// 隐含生成代码：这里只是对代码实现的建议
{noflow}
IF ptToTest=0 THEN
    ADSLOGSTR(ADSLOG_MSGTYPE_ERROR OR ADSLOG_MSGTYPE_STRING,'CheckPointer failed due to invalid address.','');
ELSIF iSize<=0 THEN
    ADSLOGSTR(ADSLOG_MSGTYPE_ERROR OR ADSLOG_MSGTYPE_STRING,'CheckPointer failed due to invalid size.','');
ELSIF iGran<=0 THEN
    ADSLOGSTR(ADSLOG_MSGTYPE_ERROR OR ADSLOG_MSGTYPE_STRING,'CheckPointer failed due to invalid granularity.','');
// -> Please note that the following memory area check is time consuming:
//ELSIF F_CheckMemoryArea(pData:=ptToTest,nSize:=DINT_TO_UDINT(iSize)) = E_TcMemoryArea.Unknown THEN
//    ADSLOGSTR(ADSLOG_MSGTYPE_ERROR OR ADSLOG_MSGTYPE_STRING,'CheckPointer failed due to unknown memory area.','');
END_IF
CheckPointer := ptToTest;
{flow}

END_FUNCTION

// ---- POUs/003_FB/43_implicit checks/CheckRangeSigned.TcPOU
// 隐含生成代码：不要编辑
FUNCTION CheckRangeSigned : DINT
VAR_INPUT
	value, lower, upper: DINT;
END_VAR

// 隐含生成代码：这里只是对代码实现的建议
{noflow}
IF (value < lower) THEN
	CheckRangeSigned := lower;
ELSIF(value > upper) THEN
	CheckRangeSigned := upper;
ELSE
	CheckRangeSigned := value;
END_IF
{flow}

END_FUNCTION

// ---- POUs/003_FB/43_implicit checks/CheckRangeUnsigned.TcPOU
// 隐含生成代码：不要编辑
FUNCTION CheckRangeUnsigned : UDINT
VAR_INPUT
	value, lower, upper: UDINT;
END_VAR

// 隐含生成代码：这里只是对代码实现的建议
{noflow}
IF (value < lower) THEN
	CheckRangeUnsigned := lower;
ELSIF(value > upper) THEN
	CheckRangeUnsigned := upper;
ELSE
	CheckRangeUnsigned := value;
END_IF
{flow}

END_FUNCTION

// ---- POUs/003_FB/53_RudongPump/08_PeristalticPumpFB/FB_RuDongPump_modbus_LABV.TcPOU
//{attribute 'tc_no_symbol'}
FUNCTION_BLOCK FB_RuDongPump_modbus_LABV
VAR_INPUT
	xExecute: BOOL;
	xAbort: BOOL;
	xResetRequest: BOOL;//匹配复位按钮 
	xRunILC				:BOOL;//蠕动泵运行条件
	dwTimeLimit: DWORD:=1;//[ms],1 => no invocation time limit
	dwTimeOut: DWORD;//[ms],0 => no executing time limit
	stPara       : RudongPump_Sys_Para;				
	xNeedConfigurePara		: BOOL := TRUE;//是否需要配置参数(默认是需要进行参数配置的)	
	stRunPara	:RudongPump_RunData;//运行参数	
	xAutoMode    : BOOL;//0:mannal 1:auto
	xIniting     : BOOL;//初始化过程中
	xDeviceRunning : BOOL;//工站单循环中
	rSpeedRatio  : REAL:=2.733;//根据泵头软管型号不同有变化
	sHmiError : STRING;
	xEStop : BOOL;
	stDeviceOpe	: RudongPump_Ope;//操作按钮
END_VAR
VAR_OUTPUT
	xDone: BOOL;(*完成条件满足*)
	xBusy: BOOL;(*动作正在执行*)
	xAborted: BOOL;(*指令被打断*)
	xRunning	:BOOL;//蠕动泵运行中
	eMobbusErrorID:UDINT;//modubs 报警信息
	xRudongPump_ERROR: BOOL;(*错误条件满足*)
	eERRORID: RudongPump_ERROR;(*错误码*)
	xRdyCmd : BOOL;
END_VAR
VAR_IN_OUT
		
END_VAR
VAR
{attribute 'tc_no_symbol'}
	eState: STATE;
{attribute 'tc_no_symbol'}
	_xDone: BOOL;
{attribute 'tc_no_symbol'}
	eCmd : RudongPump_CMD;//指令控制	
{attribute 'tc_no_symbol'}
	xFirstInvocation: BOOL := TRUE;	
{attribute 'tc_no_symbol'} 
	xTimeOut: BOOL;
{attribute 'tc_no_symbol'}
	xTimeLimit: BOOL;
{attribute 'tc_no_symbol'}
	tInvocationTimer , tOperationTimer : TON;
{attribute 'tc_no_symbol'}
	rFluVolumeSet   : REAL;//液量设定 0.0-99999.0 mL(0.1ml)
{attribute 'tc_no_symbol'}
	rRuntimeSet     : REAL;//运行时间设定 0.1-9999s(0.1s)
{attribute 'tc_no_symbol'}
	iCycleNumber		: INT;//重复次数
{attribute 'tc_no_symbol'}
	iModuleAdress		: INT;//灌装单元地址
{attribute 'tc_no_symbol'}
	iModuleSpeed		: REAL;//灌装单元速度
{attribute 'tc_no_symbol'}
	iModuleRealVolume	: REAL;//灌装实际液量	
{attribute 'tc_no_symbol'}
	_cmdStop  : BOOL;  
{attribute 'tc_no_symbol'}
	_tonTimeout , _tonCmdTimeout : TON;	
{attribute 'tc_no_symbol'}
  /// command execution
  _CmdExe : BOOL;
{attribute 'tc_no_symbol'}
  /// detect rising edge of command execution
  _rTrigCmdExe : R_TRIG;
{attribute 'tc_no_symbol'}	
  _rTrigCmdOrg   : R_TRIG;	
{attribute 'tc_no_symbol'}
	_diCmdState 	: DINT; 
{attribute 'tc_no_symbol'} 
  /// detect FltQuit rising edge
  _rTrigFltReset      : R_TRIG; 
{attribute 'tc_no_symbol'} 
  _tonDelay : TON; 
{attribute 'tc_no_symbol'}	
	_iConnectState : INT := 0;
{attribute 'tc_no_symbol'}	
	_connectTon : TON;
{attribute 'tc_no_symbol'}		
	_xConnectError : BOOL;
{attribute 'tc_no_symbol'}		
	_fResetCheck : F_TRIG;
{attribute 'tc_no_symbol'}		
	_rManual : R_TRIG;
{attribute 'tc_no_symbol'}		
	_fManual : F_TRIG;
{attribute 'tc_no_symbol'}		
	_xModeChange : BOOL;
{attribute 'tc_no_symbol'}		
	i : INT;
{attribute 'tc_no_symbol'}		
	_tonPulse : TON;//状态读取计时定时器
{attribute 'tc_no_symbol'}		
  _xCheckModbusRun : BOOL;//检测modbus是否处理总
{attribute 'tc_no_symbol'}	  
	_xConfigureParaOK : BOOL;//需要匹配参数是OK的
{attribute 'tc_no_symbol'}		
	_rStopCmdTrig : R_TRIG;
{attribute 'tc_no_symbol'}		
	_iActRunNumber : INT ;//当前运行的次数
{attribute 'tc_no_symbol'}		
	_wFluVolumeSetTemp : WORD;
{attribute 'tc_no_symbol'}		
	_wRuntimeSetTemp : WORD;
{attribute 'tc_no_symbol'}		
	_wSpeedSetTemp : WORD;	
{attribute 'tc_no_symbol'}	
 _tonDelay1:TON;
{attribute 'tc_no_symbol'}		
	_rSetSpeed : REAL;
{attribute 'tc_no_symbol'}		
	_wModuleSpeedSetTemp:WORD;
{attribute 'tc_no_symbol'}		
	_wModuleRealVolumeTemp:WORD;
{attribute 'tc_no_symbol'}		
	_rHMIControl : R_TRIG;
{attribute 'tc_no_symbol'}
	_iComNGCount:INT;
{attribute 'tc_no_symbol'}		
	dwTest1 : DWORD ;
{attribute 'tc_no_symbol'}		
	_iNGCount : INT;//NG 计数
{attribute 'tc_no_symbol'}		
	_rOperaTrig	:ARRAY [1..15] OF R_TRIG;
{attribute 'tc_no_symbol'}		
	k : INT;
{attribute 'tc_no_symbol'}		
	_bChannelNum , _bDiagData : BYTE;
{attribute 'tc_no_symbol'}		
	xAutomodeFlag	:BOOL;
{attribute 'tc_no_symbol'}		
	diStepOld:DINT;
{attribute 'tc_no_symbol'}			
	st_IOData : RudongPump_IOData;
{attribute 'tc_no_symbol'}		
	iPumpType	:INT;
{attribute 'tc_no_symbol'}	
	_xHMIOpe :BOOL;//是否有手动操作，是否有自动操作	
{attribute 'tc_no_symbol'}	
	 _xAutoOpe : BOOL;//是否有手动操作，是否有自动操作	
{attribute 'tc_no_symbol'}	
	_rInit	:R_TRIG;
{attribute 'tc_no_symbol'}		
	_first:BOOL;
{attribute 'tc_no_symbol'}				
	_aWrite_VAR: FB_MBWriteRegs; 
{attribute 'tc_no_symbol'}
//1:泵头型号；2:软管型号；3:启停控制	4:方向控制  5:全速运行  6:设定液量  7:时间设定  8:运行模式  9:重复次数		
//10:灌装单元地址  11:灌装单元速度  12:灌装单元启停  13:实际灌装量  14:灌装液量微调  15:恢复校准系数 			
  _aExecute : ARRAY[1..15] OF BOOL;    
{attribute 'tc_no_symbol'}	
  _aQuantity : ARRAY[1..15] OF WORD:=[1,1,1,1,1,2,2,1,1,1,2,1,2,1,1];  //寄存器个数   
{attribute 'tc_no_symbol'}	
  _aMBAddr : ARRAY[1..15] OF WORD:=[1000,1001,1008,1009,1010,1015,1018,1020,1023,2000,2001,2003,2004,2006,2007];  //起始地址   
{attribute 'tc_no_symbol'}		
  _aAddr : ARRAY[1..15,1..2] OF  INT;  //存放区域  
{attribute 'tc_no_symbol'}		
	_iChannelIndex:INT;
{attribute 'tc_no_symbol'}	
	_rxState:INT;
{attribute 'tc_no_symbol'}			
	_xBusy:BOOL;
END_VAR
VAR_TEMP
{attribute 'tc_no_symbol'}	
	xAgain: BOOL;
END_VAR

xAgain:=0;
ConnectAction();//触发通信连接功能连接
ACTMap();//IO Map
IF NOT _first THEN
	_first:=TRUE;
ELSE

//只有在运行的时候，才会检测是否有模式切换发生
IF eState <> STATE.DORMANT
THEN	
	IF _rManual.Q OR _fManual.Q
	THEN
		_xModeChange := TRUE;//通知系统有模式切换发生
	END_IF
ELSE
	_xModeChange := FALSE;//待机状态不触发模式切换
END_IF

//检测是否是初始化中，如果是的去切换模式
_rInit(CLK:= xIniting);
IF _rInit.Q
THEN
	eState := STATE.RESETING;
END_IF	

REPEAT
	CASE eState OF
		STATE.DORMANT:
				HandleDormantState(xAgain=> xAgain);
		STATE.EXECUTING:
				HandleExecutingState(xAgain=> xAgain);
		STATE.DONE:
				HandleDoneState(xAgain=> xAgain);
		STATE.INERROR:
				HandleErrorState(xAgain=> xAgain);
		STATE.ABORTING:
				HandleAbortingState(xAgain=> xAgain);
		STATE.ABORTED:
				HandleAbortedState(xAgain=> xAgain);
		STATE.RESETING:
				HandleResettingState(xAgain=> xAgain);
	END_CASE
UNTIL (xAgain=0)
END_REPEAT
END_IF


//判断是否处于当前流程的Done状态
xDone := _xDone AND xExecute;
//输出报错信息
CASE eERRORID OF 	
  RudongPump_ERROR.No_ERROR:
		sHmiError:='No_ERROR';	
  RudongPump_ERROR.FLT_PARA:
		sHmiError:='FLT_PARA';
  RudongPump_ERROR.FLT_CONNECT:
		sHmiError:='FLT_CONNECT';
  RudongPump_ERROR.FLT_RDYCMD:
		sHmiError:='FLT_RDYCMD';
	RudongPump_ERROR.FLT_CONFIGURE_PARA:
		sHmiError:='FLT_CONFIGURE_PARA';
	RudongPump_ERROR.FLT_FLUVOLUM_TIME_PARA:
		sHmiError:='FLT_FLUVOLUM_TIME_PARA';  
  RudongPump_ERROR.FLT_PUSH_TIMEOUT:
		sHmiError:='FLT_PUSH_TIMEOUT';
  RudongPump_ERROR.FLT_PULL_TIMEOUT:
		sHmiError:='FLT_PULL_TIMEOUT';
  RudongPump_ERROR.FLT_STOP_TIMEOUT:
		sHmiError:='FLT_STOP_TIMEOUT'; 
	RudongPump_ERROR.FLT_FULLSPEEDSTOP_TIMEOUT:
		sHmiError:='FLT_FULLSPEEDSTOP_TIMEOUT';
	RudongPump_ERROR.FLT_FULLSPEEDSTART_TIMEOUT:
		sHmiError:='FLT_FULLSPEEDSTART_TIMEOUT'; 
	RudongPump_ERROR.FLT_CMD_TIMEOUT:
		sHmiError:='FLT_CMD_TIMEOUT';
	RudongPump_ERROR.FLT_RUN_FALL:
		sHmiError:='FLT_RUN_FALL';
END_CASE
//手动自动操作检测
_xHMIOpe :=
			stDeviceOpe.xConfigure_Hmi OR 
			stDeviceOpe.xFullSpeedPull_Hmi OR 
			stDeviceOpe.xFullSpeedPush_Hmi OR 
			stDeviceOpe.xPull_Hmi[1] OR 
			stDeviceOpe.xPull_Hmi[2] OR 
			stDeviceOpe.xPull_Hmi[3] OR 
			stDeviceOpe.xPull_Hmi[4] OR 
			stDeviceOpe.xPull_Hmi[5] OR 			
			stDeviceOpe.xPumpCal_Hmi OR 
			stDeviceOpe.xPush_Hmi[1] OR 
			stDeviceOpe.xPush_Hmi[2] OR 
			stDeviceOpe.xPush_Hmi[3] OR 			
			stDeviceOpe.xPush_Hmi[4] OR 			
			stDeviceOpe.xPush_Hmi[5] OR 						
			stDeviceOpe.xResetCalcoeffCal_Hmi OR 
			stDeviceOpe.xStop_Hmi;
_xAutoOpe:=	
			stDeviceOpe.xConfigure_Auto OR 
            stDeviceOpe.xFullSpeedPull_Auto OR 
            stDeviceOpe.xFullSpeedPush_Auto OR 
            stDeviceOpe.xPull_Auto[1] OR 
            stDeviceOpe.xPull_Auto[2] OR 			
            stDeviceOpe.xPull_Auto[3] OR 			
            stDeviceOpe.xPull_Auto[4] OR 			
            stDeviceOpe.xPull_Auto[5] OR 			
            stDeviceOpe.xPumpCal_Auto OR 
            stDeviceOpe.xPush_Auto[1] OR 
            stDeviceOpe.xPush_Auto[2] OR 			
            stDeviceOpe.xPush_Auto[3] OR 			
            stDeviceOpe.xPush_Auto[4] OR 			
            stDeviceOpe.xPush_Auto[5] OR 						
            stDeviceOpe.xStop_Auto;

METHOD PROTECTED AbortAction
VAR_INPUT
END_VAR
VAR_OUTPUT
	xComplete: BOOL;
  eERRORID: RudongPump_ERROR;
END_VAR
(*
* Cleaning
* => abort all running operation
* => if an NBS.RudongPump_ERROR codition is reached, set eERRORID to a Value rather then NBS.RudongPump_ERROR.No_ERROR 
*)
xComplete:=1;
eERRORID:=RudongPump_ERROR.No_ERROR;
END_METHOD

ACTION ACTMap:

//1,泵头类型
	_aAddr[1,1]:= st_IOData.O_PumpType;
//2,软管类型	
	_aAddr[2,1] := st_IOData.O_HosePipeType;
//3,启停控制	
	_aAddr[3,1] := st_IOData.O_ControlSet;
//4,方向控制	
	_aAddr[4,1] := st_IOData.O_DirectionSet;
//5,全速控制	
	_aAddr[5,1] := st_IOData.O_FullSpeedControl;	
//6,液量设定	
	SysMemCpy(ADR(_aAddr[6,1]),ADR(st_IOData.O_FluVolumeSet),4);	
	_wFluVolumeSetTemp := TO_WORD(_aAddr[6,1]);
	_aAddr[6,1] := _aAddr[6,2];
	_aAddr[6,2] := TO_INT(_wFluVolumeSetTemp);
//7,运行时间设定	
	SysMemCpy(ADR(_aAddr[7,1]),ADR(st_IOData.O_RuntimeSet),4);
	_wRuntimeSetTemp := TO_WORD(_aAddr[7,1]);
	_aAddr[7,1] := _aAddr[7,2];
	_aAddr[7,2] := TO_INT(_wRuntimeSetTemp);	
//8,运行模式	
	_aAddr[8,1] := st_IOData.O_RunModeSet;
//9,重复次数	
	_aAddr[9,1] := st_IOData.O_CycleNumber;
//10,灌装单元地址
	_aAddr[10,1] := st_IOData.O_ModuleAddress;	
//11,灌装单元速度
	SysMemCpy(ADR(_aAddr[11,1]),ADR(st_IOData.O_ModuleSpeed),4);
	_wModuleSpeedSetTemp := TO_WORD(_aAddr[11,1]);
	_aAddr[11,1] := _aAddr[11,2];
	_aAddr[11,2] := TO_INT(_wModuleSpeedSetTemp);
//12,灌装单元启停
	_aAddr[12,1] := st_IOData.O_ModuleStart;	
//13,实际灌装液量
	SysMemCpy(ADR(_aAddr[13,1]),ADR(st_IOData.O_ModuleRealVolume),4);
	_wModuleRealVolumeTemp := TO_WORD(_aAddr[13,1]);
	_aAddr[13,1] := _aAddr[13,2];
	_aAddr[13,2] := TO_INT(_wModuleRealVolumeTemp);
//14,灌装液量微调
	_aAddr[14,1] := st_IOData.O_ModuleMicroReg;	
//15,恢复校准系数
	_aAddr[15,1] := st_IOData.O_ResetCalcoeff;		

xRunning:=stPara.xPumpRunSignal;//运行信号
iPumpType:=RudongPump_PumpType.LabV;//蠕动泵类型

_fResetCheck(CLK:=xResetRequest);
xRdyCmd := eState = STATE.DORMANT AND eERRORID = RudongPump_ERROR.No_ERROR;//检测是否允许指令控制(初始状态，没有报警发生)
(**********************************检测是否有模式切换********************************)
_rManual(CLK:=xAutoMode);
_fManual(CLK:=xAutoMode);
IF eState <> STATE.DORMANT//只有在运行的时候，才会检测是否有模式切换发生
THEN
	IF _rManual.Q OR _fManual.Q
	THEN
		_xModeChange := TRUE;//通知系统有模式切换发生
	END_IF	
END_IF
IF eState = STATE.DORMANT//要是待机模式下，切换模式，是不会起作用的
THEN
	_xModeChange := FALSE;
END_IF
(*************************检测配置参数是否匹配成功*********************************)
IF ( ( stRunPara.iPumpTypeSet = 0 OR stRunPara.iPumpTypeSet = 2 ) AND ( ( stRunPara.iHosePipeTypeSet >=13 AND stRunPara.iHosePipeTypeSet <=14 ) OR  
	 ( stRunPara.iHosePipeTypeSet >= 16 AND stRunPara.iHosePipeTypeSet <= 19 ) OR  stRunPara.iHosePipeTypeSet = 25 )) OR 
	 ( ( stRunPara.iPumpTypeSet = 1 OR stRunPara.iPumpTypeSet =3 ) AND ( stRunPara.iHosePipeTypeSet = 15 OR stRunPara.iHosePipeTypeSet = 24 ) ) OR 
	 ( ( stRunPara.iPumpTypeSet = 4 OR stRunPara.iPumpTypeSet = 5 ) AND (stRunPara.iHosePipeTypeSet >= 101 AND stRunPara.iHosePipeTypeSet <= 105 )) OR 
	 ( stRunPara.iPumpTypeSet = 6 AND (stRunPara.iHosePipeTypeSet = 15 OR stRunPara.iHosePipeTypeSet = 24 OR stRunPara.iHosePipeTypeSet = 35 OR stRunPara.iHosePipeTypeSet = 36)) OR 
	 ( stRunPara.iPumpTypeSet = 7 AND ( stRunPara.iHosePipeTypeSet = 14 OR stRunPara.iHosePipeTypeSet = 16 )) OR 
	 ( stRunPara.iPumpTypeSet = 8 AND stRunPara.iHosePipeTypeSet = 24 ) OR
   ( stRunPara.iPumpTypeSet = 17 AND (stRunPara.iHosePipeTypeSet = 15 OR stRunPara.iHosePipeTypeSet = 24 OR stRunPara.iHosePipeTypeSet = 35 OR stRunPara.iHosePipeTypeSet = 36) )	 
THEN
  _xConfigureParaOK := TRUE;
ELSE
	_xConfigureParaOK := FALSE;
END_IF
END_ACTION

METHOD PROTECTED CmdCalReset
VAR_OUTPUT
	xComplete: BOOL;
END_VAR
// return the real actual fault number
IF eERRORID <> RudongPump_ERROR.No_ERROR
THEN
  RETURN;  
END_IF

CASE _diCmdState OF	
		
		
	0://发送灌装系数复位指令
		_tonDelay(IN:= TRUE,pt:=T#20MS);//保证执行的是最新的一次
		st_IOData.O_ResetCalcoeff := 1	;	
		IF _tonDelay.Q
		THEN	
			_aExecute[15] := TRUE;//	
			//复位定时器
			_tonDelay(IN:=FALSE);
			_tonCmdTimeout(in:=FALSE);
			_tonTimeout(in:=FALSE);
			_diCmdState := _diCmdState+1;//切换状态
		END_IF
		
	1://等待灌装启动被响应
		_tonCmdTimeout(IN:= _aExecute[15],pt:=T#2S);
		IF NOT _aExecute[15]//
		THEN		
			_tonDelay(IN:=TRUE,PT:= T#50MS);
			IF _tonDelay.Q
			THEN
				_tonTimeout(in:=FALSE);
				_tonDelay(IN:=FALSE);
				_tonCmdTimeout(IN:= FALSE); 
				_diCmdState := _diCmdState+1;//切换状态
			END_IF	
		END_IF	
		IF _tonCmdTimeout.Q
		THEN
			eERRORID := RudongPump_ERROR.FLT_CMD_TIMEOUT;		
			_diCmdState := 999;
		END_IF	

	2://
		xComplete := TRUE; 
		
	ELSE
		;	
END_CASE
END_METHOD

METHOD PROTECTED CmdPumpCal
VAR_OUTPUT
	xComplete: BOOL;
END_VAR
// return the real actual fault number
IF eERRORID <> RudongPump_ERROR.No_ERROR
THEN
  RETURN;  
END_IF

CASE _diCmdState OF	
	0://检查参数	  	
		IF xNeedConfigurePara
		THEN
			_tonDelay(IN:= TRUE,pt:=T#25MS);//保证执行的是最新的一次
			st_IOData.O_RunModeSet := 2	;//打开定时定量模式
			IF _tonDelay.Q
			THEN	
				_aExecute[8] := TRUE;//启动夹紧控制数据发送	
				//复位定时器
				_tonDelay(IN:=FALSE);
				_tonCmdTimeout(in:=FALSE);
				_tonTimeout(in:=FALSE);
				_diCmdState := _diCmdState+1;//切换状态
			END_IF
		ELSE//直接启动就好
			//复位定时器
			_tonDelay(IN:=FALSE);
			_tonCmdTimeout(in:=FALSE);
			_tonTimeout(in:=FALSE);
			_diCmdState := 8;//切换状态
		END_IF	
		//检测流量转速是否在0.1rpm - 600rpm
		IF 	rRuntimeSet = 0 
		THEN 
			eERRORID := RudongPump_ERROR.FLT_FLUVOLUM_TIME_PARA;		
			_diCmdState := 999;
		ELSE
			_rSetSpeed := rFluVolumeSet * 60.0 / rSpeedRatio / rRuntimeSet;
			IF _rSetSpeed >= 0.1 AND _rSetSpeed <= 600
			THEN
				;
			ELSE
				eERRORID := RudongPump_ERROR.FLT_FLUVOLUM_TIME_PARA;		
				_diCmdState := 999;
			END_IF
		END_IF				
		
	1://等待定时定量模式被响应
		_tonCmdTimeout(IN:= _aExecute[8],pt:=T#2S);
		IF NOT _aExecute[8]//
		THEN		
			_tonDelay(IN:=TRUE,PT:= T#50MS);
			IF _tonDelay.Q
			THEN			
				_tonTimeout(in:=FALSE);
				_tonDelay(IN:=FALSE);
				_tonCmdTimeout(IN:= FALSE);    
				_diCmdState := _diCmdState+1;//切换状态
			END_IF	
		END_IF	
		IF _tonCmdTimeout.Q
		THEN
			eERRORID := RudongPump_ERROR.FLT_CMD_TIMEOUT;		
			_diCmdState := 999;
		END_IF


//发送虚假定量时间		
	2://定量时间设定		
		_tonDelay(IN:= TRUE,pt:=T#25MS);//保证执行的是最新的一次
		st_IOData.O_RuntimeSet := 200.0	;	//保证电机转速不会超
		IF _tonDelay.Q
		THEN	
			_aExecute[7] := TRUE;//启动夹紧控制数据发送	
			//复位定时器
			_tonDelay(IN:=FALSE);
			_tonCmdTimeout(in:=FALSE);
			_tonTimeout(in:=FALSE);
			_diCmdState := _diCmdState+1;//切换状态
		END_IF
	3://等待定量时间设定被响应
		_tonCmdTimeout(IN:= _aExecute[7],pt:=T#2S);
		IF NOT _aExecute[7]//
		THEN		
			_tonDelay(IN:=TRUE,PT:= T#50MS);
			IF _tonDelay.Q
			THEN			
				_tonTimeout(in:=FALSE);
				_tonDelay(IN:=FALSE);
				_tonCmdTimeout(IN:= FALSE);    
				_diCmdState := _diCmdState+1;//切换状态
			END_IF	
		END_IF	
		IF _tonCmdTimeout.Q
		THEN
			eERRORID := RudongPump_ERROR.FLT_CMD_TIMEOUT;		
			_diCmdState := 999;
		END_IF		
		
		
//传递液量参数		
	4://		
		_tonDelay(IN:= TRUE,pt:=T#25MS);//保证执行的是最新的一次
		st_IOData.O_FluVolumeSet := rFluVolumeSet	;	
		IF _tonDelay.Q
		THEN	
			_aExecute[6] := TRUE;//启动夹紧控制数据发送	
			//复位定时器
			_tonDelay(IN:=FALSE);
			_tonCmdTimeout(in:=FALSE);
			_tonTimeout(in:=FALSE);
			_diCmdState := _diCmdState+1;//切换状态
		END_IF	  
	5://等待流量设定结束
		_tonCmdTimeout(IN:= _aExecute[6],pt:=T#2S);
		IF NOT _aExecute[6]//
		THEN		
			_tonDelay(IN:=TRUE,PT:= T#50MS);
			IF _tonDelay.Q
			THEN			
				_tonTimeout(in:=FALSE);
				_tonDelay(IN:=FALSE);
				_tonCmdTimeout(IN:= FALSE);    
				_diCmdState := _diCmdState+1;//切换状态
			END_IF	
		END_IF	
		IF _tonCmdTimeout.Q
		THEN
			eERRORID := RudongPump_ERROR.FLT_CMD_TIMEOUT;		
			_diCmdState := 999;
		END_IF

//传递实际定量时间		
	6://定量时间设定		
		_tonDelay(IN:= TRUE,pt:=T#25MS);//保证执行的是最新的一次
		st_IOData.O_RuntimeSet := rRuntimeSet	;	
		IF _tonDelay.Q
		THEN	
			_aExecute[7] := TRUE;//启动夹紧控制数据发送	
			//复位定时器
			_tonDelay(IN:=FALSE);
			_tonCmdTimeout(in:=FALSE);
			_tonTimeout(in:=FALSE);
			_diCmdState := _diCmdState+1;//切换状态
		END_IF
		
	7://等待定量时间设定被响应
		_tonCmdTimeout(IN:= _aExecute[7],pt:=T#2S);
		IF NOT _aExecute[7]//
		THEN		
			_tonDelay(IN:=TRUE,PT:= T#50MS);
			IF _tonDelay.Q
			THEN			
				_tonTimeout(in:=FALSE);
				_tonDelay(IN:=FALSE);
				_tonCmdTimeout(IN:= FALSE);    
				_diCmdState := _diCmdState+1;//切换状态
			END_IF	
		END_IF	
		IF _tonCmdTimeout.Q
		THEN
			eERRORID := RudongPump_ERROR.FLT_CMD_TIMEOUT;		
			_diCmdState := 999;
		END_IF	
		
	8://方向设定		
		_tonDelay(IN:= ( eCmd = RudongPump_CMD.Cmd_CalPump ) ,pt:=T#20MS);//保证执行的是最新的一次
		st_IOData.O_DirectionSet := 1	;			
		IF _tonDelay.Q
		THEN	
			_aExecute[4] := TRUE;//启动夹紧控制数据发送	
			//复位定时器
			_tonDelay(IN:=FALSE);
			_tonCmdTimeout(in:=FALSE);
			_tonTimeout(in:=FALSE);
			_diCmdState := _diCmdState+1;//切换状态
		END_IF
		
	9://等待方向设定被响应
		_tonCmdTimeout(IN:= _aExecute[4],pt:=T#2S);
		IF NOT _aExecute[4]//
		THEN		
			_diCmdState := _diCmdState +1; 
			_tonDelay(IN:=FALSE);
			_tonCmdTimeout(in:=FALSE);
			_tonTimeout(in:=FALSE);
		END_IF	
		IF _tonCmdTimeout.Q
		THEN
			eERRORID := RudongPump_ERROR.FLT_CMD_TIMEOUT;		
			_diCmdState := 999;
		END_IF	
		
	10://重复次数设定		
		_tonDelay(IN:= TRUE,pt:=T#25MS);//保证执行的是最新的一次
		st_IOData.O_CycleNumber := iCycleNumber	;	
		IF _tonDelay.Q
		THEN	
			_aExecute[9] := TRUE;//启动夹紧控制数据发送	
			//复位定时器
			_tonDelay(IN:=FALSE);
			_tonCmdTimeout(in:=FALSE);
			_tonTimeout(in:=FALSE);
			_diCmdState := _diCmdState+1;//切换状态
		END_IF
		
	11://等待重复次数设定被响应
		_tonCmdTimeout(IN:= _aExecute[9],pt:=T#2S);
		IF NOT _aExecute[9]//
		THEN		
			_tonDelay(IN:=TRUE,PT:= T#50MS);
			IF _tonDelay.Q
			THEN
				_tonTimeout(in:=FALSE);
				_tonDelay(IN:=FALSE);
				_tonCmdTimeout(IN:= FALSE); 
				_diCmdState := _diCmdState+1;//切换状态
			END_IF	
		END_IF	
		IF _tonCmdTimeout.Q
		THEN
			eERRORID := RudongPump_ERROR.FLT_CMD_TIMEOUT;		
			_diCmdState := 999;
		END_IF		
		
	12://单元地址设定
		_tonDelay(IN:= TRUE,pt:=T#20MS);//保证执行的是最新的一次
		st_IOData.O_ModuleAddress := iModuleAdress	;
		//st_IOData.O_ModuleSpeed := iModuleSpeed	;	
		IF _tonDelay.Q
		THEN	
			_aExecute[10] := TRUE;//	
			//复位定时器
			_tonDelay(IN:=FALSE);
			_tonCmdTimeout(in:=FALSE);
			_tonTimeout(in:=FALSE);
			_diCmdState := _diCmdState+1;//切换状态
		END_IF
		
	13://等待单元地址设定被响应
	IF iPumpType=RudongPump_PumpType.DFPluse THEN	
		_tonCmdTimeout(IN:= _aExecute[10],pt:=T#2S);
		IF NOT _aExecute[10]//
		THEN		
			_tonDelay(IN:=TRUE,PT:= T#50MS);
			IF _tonDelay.Q
			THEN
				_tonTimeout(in:=FALSE);
				_tonDelay(IN:=FALSE);
				_tonCmdTimeout(IN:= FALSE); 
				_diCmdState := _diCmdState+1;//切换状态
			END_IF	
		END_IF	
		IF _tonCmdTimeout.Q
		THEN
			eERRORID := RudongPump_ERROR.FLT_CMD_TIMEOUT;		
			_diCmdState := 999;
		END_IF
	ELSE
		_diCmdState := 15;	
	END_IF	
		
	14://单元速度设定
	IF st_IOData.O_RunModeSet =1	THEN//如果是定量模式，需要设置速度
		_tonDelay(IN:= TRUE,pt:=T#20MS);//保证执行的是最新的一次
		st_IOData.O_ModuleSpeed := iModuleSpeed	;	
		IF _tonDelay.Q
		THEN	
			_aExecute[11] := TRUE;//	
			//复位定时器
			_tonDelay(IN:=FALSE);
			_tonCmdTimeout(in:=FALSE);
			_tonTimeout(in:=FALSE);
			_diCmdState := _diCmdState+1;//切换状态
		END_IF
	ELSE
		_diCmdState :=16;//如果是定时定量模式，则不需要设置速度
	END_IF	
	
	15://等待单元速度设定被响应
		_iNGCount :=0;
		_tonCmdTimeout(IN:= _aExecute[11],pt:=T#2S);
		IF NOT _aExecute[11]//
		THEN		
			_tonDelay(IN:=TRUE,PT:= T#50MS);
			IF _tonDelay.Q
			THEN
				_tonTimeout(in:=FALSE);
				_tonDelay(IN:=FALSE);
				_tonCmdTimeout(IN:= FALSE); 
				_diCmdState := _diCmdState+1;//切换状态
			END_IF	
		END_IF	
		IF _tonCmdTimeout.Q
		THEN
			eERRORID := RudongPump_ERROR.FLT_CMD_TIMEOUT;		
			_diCmdState := 999;
		END_IF		
		
	16://复位	
		st_IOData.O_ModuleStart := 0	;
		_aExecute[12] := FALSE;//		
		_diCmdState := _diCmdState+1;//切换状态
		
	17://灌装启动
		_tonDelay(IN:= TRUE,pt:=T#20MS);//保证执行的是最新的一次
		st_IOData.O_ModuleStart := 1	;	
		IF _tonDelay.Q
		THEN	
			_aExecute[12] := TRUE;//	
			//复位定时器
			_tonDelay(IN:=FALSE);
			_tonCmdTimeout(in:=FALSE);
			_tonTimeout(in:=FALSE);
			_diCmdState := _diCmdState+1;//切换状态
		END_IF
		
	18://等待灌装启动被响应
		_tonTimeout(in:=TRUE,pt:=T#30MS); 		
		_tonCmdTimeout(IN:= _aExecute[12],pt:=T#2S);
		IF stPara.xPumpRunSignal//一定要检测到泵运行
		THEN		
			_tonDelay(IN:=FALSE);
			_tonCmdTimeout(in:=FALSE);
			_diCmdState := _diCmdState +1; 
			_tonTimeout(in:=FALSE);	
		END_IF			
		IF _tonCmdTimeout.Q
		THEN
			eERRORID := RudongPump_ERROR.FLT_CMD_TIMEOUT;		
			_diCmdState := 999;
		END_IF
	IF _tonCmdTimeout.Q THEN
		_iNGCount := _iNGCount + 1;		
		IF _iNGCount <= 3
		THEN
			_tonDelay(IN:=FALSE);
			_tonCmdTimeout(IN:=FALSE);
			_tonTimeout(IN:=FALSE);
			_diCmdState := 15;//重新触发启动
		ELSE
			eERRORID := RudongPump_ERROR.FLT_PumpCal_TIMEOUT;					
			_diCmdState := 999;
		END_IF
	 END_IF		
		
	19://等待接液完成
		IF NOT stPara.xPumpRunSignal AND (stDeviceOpe.xPumpCal_Hmi OR stDeviceOpe.xPumpCal_Auto) AND NOT _xCheckModbusRun THEN
			_diCmdState := _diCmdState+1;//切换状态
		END_IF
		
	20://单元实际液量设定
		_tonDelay(IN:= TRUE,pt:=T#20MS);//保证执行的是最新的一次
		st_IOData.O_ModuleRealVolume := iModuleRealVolume	;	
		IF _tonDelay.Q
		THEN	
			_aExecute[13] := TRUE;//	
			//复位定时器
			_tonDelay(IN:=FALSE);
			_tonCmdTimeout(in:=FALSE);
			_tonTimeout(in:=FALSE);
			_diCmdState := _diCmdState+1;//切换状态
		END_IF
		
	21://等待单元实际液量设定被响应
		_tonCmdTimeout(IN:= _aExecute[13],pt:=T#2S);
		IF NOT _aExecute[13]//
		THEN		
			_tonDelay(IN:=TRUE,PT:= T#50MS);
			IF _tonDelay.Q
			THEN
				_tonTimeout(in:=FALSE);
				_tonDelay(IN:=FALSE);
				_tonCmdTimeout(IN:= FALSE); 
				_diCmdState := _diCmdState+1;//切换状态
			END_IF	
		END_IF	
		IF _tonCmdTimeout.Q
		THEN
			eERRORID := RudongPump_ERROR.FLT_CMD_TIMEOUT;		
			_diCmdState := 999;
		END_IF		

	22://
		xComplete := TRUE; 
		
	ELSE
		;	
END_CASE
END_METHOD

METHOD PROTECTED CmdRunAction
VAR_OUTPUT
	xComplete: BOOL;
END_VAR
// return the real actual fault number
IF eERRORID <> RudongPump_ERROR.No_ERROR
THEN
  RETURN;  
END_IF

CASE _diCmdState OF	
	0://传送力值和速度参数		  	
		IF xNeedConfigurePara
		THEN
			_tonDelay(IN:= TRUE,pt:=T#25MS);//保证执行的是最新的一次
			st_IOData.O_RunModeSet := 2	;//打开定时定量模式
			IF _tonDelay.Q
			THEN	
				_aExecute[8] := TRUE;//启动夹紧控制数据发送	
				//复位定时器
				_tonDelay(IN:=FALSE);
				_tonCmdTimeout(in:=FALSE);
				_tonTimeout(in:=FALSE);
				_diCmdState := _diCmdState+1;//切换状态
			END_IF
		ELSE//直接启动就好
			//复位定时器
			_tonDelay(IN:=FALSE);
			_tonCmdTimeout(in:=FALSE);
			_tonTimeout(in:=FALSE);
			_diCmdState := 12;//切换状态
		END_IF	
		//检测流量转速是否在0.1rpm - 600rpm
		IF 	rRuntimeSet = 0 
		THEN 
			eERRORID := RudongPump_ERROR.FLT_FLUVOLUM_TIME_PARA;		
			_diCmdState := 999;
		ELSE
			_rSetSpeed := rFluVolumeSet * 60.0 / rSpeedRatio / rRuntimeSet;
			IF _rSetSpeed >= 0.1 AND _rSetSpeed <= 600
			THEN
				;
			ELSE
				eERRORID := RudongPump_ERROR.FLT_FLUVOLUM_TIME_PARA;		
				_diCmdState := 999;
			END_IF
		END_IF				
		
	1://等待定时定量模式被响应
		_tonCmdTimeout(IN:= _aExecute[8],pt:=T#2S);
		IF NOT _aExecute[8]//
		THEN		
			_tonDelay(IN:=TRUE,PT:= T#50MS);
			IF _tonDelay.Q
			THEN			
				_tonTimeout(in:=FALSE);
				_tonDelay(IN:=FALSE);
				_tonCmdTimeout(IN:= FALSE);    
				_diCmdState := _diCmdState+1;//切换状态
			END_IF	
		END_IF	
		IF _tonCmdTimeout.Q
		THEN
			eERRORID := RudongPump_ERROR.FLT_CMD_TIMEOUT;		
			_diCmdState := 999;
		END_IF


//发送虚假定量时间		
	2://定量时间设定		
		_tonDelay(IN:= TRUE,pt:=T#25MS);//保证执行的是最新的一次
		st_IOData.O_RuntimeSet := 200.0	;	//保证电机转速不会超
		IF _tonDelay.Q
		THEN	
			_aExecute[7] := TRUE;//启动夹紧控制数据发送	
			//复位定时器
			_tonDelay(IN:=FALSE);
			_tonCmdTimeout(in:=FALSE);
			_tonTimeout(in:=FALSE);
			_diCmdState := _diCmdState+1;//切换状态
		END_IF
	3://等待定量时间设定被响应
		_tonCmdTimeout(IN:= _aExecute[7],pt:=T#2S);
		IF NOT _aExecute[7]//
		THEN		
			_tonDelay(IN:=TRUE,PT:= T#50MS);
			IF _tonDelay.Q
			THEN			
				_tonTimeout(in:=FALSE);
				_tonDelay(IN:=FALSE);
				_tonCmdTimeout(IN:= FALSE);    
				_diCmdState := _diCmdState+1;//切换状态
			END_IF	
		END_IF	
		IF _tonCmdTimeout.Q
		THEN
			eERRORID := RudongPump_ERROR.FLT_CMD_TIMEOUT;		
			_diCmdState := 999;
		END_IF		
		
		
//传递液量参数		
	4://传送力值和速度参数		
		_tonDelay(IN:= TRUE,pt:=T#25MS);//保证执行的是最新的一次
		st_IOData.O_FluVolumeSet := rFluVolumeSet	;	
		IF _tonDelay.Q
		THEN	
			_aExecute[6] := TRUE;//启动夹紧控制数据发送	
			//复位定时器
			_tonDelay(IN:=FALSE);
			_tonCmdTimeout(in:=FALSE);
			_tonTimeout(in:=FALSE);
			_diCmdState := _diCmdState+1;//切换状态
		END_IF	  
	5://等待流量设定结束
		_tonCmdTimeout(IN:= _aExecute[6],pt:=T#2S);
		IF NOT _aExecute[6]//
		THEN		
			_tonDelay(IN:=TRUE,PT:= T#50MS);
			IF _tonDelay.Q
			THEN			
				_tonTimeout(in:=FALSE);
				_tonDelay(IN:=FALSE);
				_tonCmdTimeout(IN:= FALSE);    
				_diCmdState := _diCmdState+1;//切换状态
			END_IF	
		END_IF	
		IF _tonCmdTimeout.Q
		THEN
			eERRORID := RudongPump_ERROR.FLT_CMD_TIMEOUT;		
			_diCmdState := 999;
		END_IF

//传递实际定量时间		
	6://定量时间设定		
		_tonDelay(IN:= TRUE,pt:=T#25MS);//保证执行的是最新的一次
		st_IOData.O_RuntimeSet := rRuntimeSet	;	
		IF _tonDelay.Q
		THEN	
			_aExecute[7] := TRUE;//启动夹紧控制数据发送	
			//复位定时器
			_tonDelay(IN:=FALSE);
			_tonCmdTimeout(in:=FALSE);
			_tonTimeout(in:=FALSE);
			_diCmdState := _diCmdState+1;//切换状态
		END_IF
		
	7://等待定量时间设定被响应
		_tonCmdTimeout(IN:= _aExecute[7],pt:=T#2S);
		IF NOT _aExecute[7]//
		THEN		
			_tonDelay(IN:=TRUE,PT:= T#50MS);
			IF _tonDelay.Q
			THEN			
				_tonTimeout(in:=FALSE);
				_tonDelay(IN:=FALSE);
				_tonCmdTimeout(IN:= FALSE);    
				_diCmdState := _diCmdState+1;//切换状态
			END_IF	
		END_IF	
		IF _tonCmdTimeout.Q
		THEN
			eERRORID := RudongPump_ERROR.FLT_CMD_TIMEOUT;		
			_diCmdState := 999;
		END_IF	
		
	8://方向设定		
		_tonDelay(IN:= ( eCmd = RudongPump_CMD.Cmd_Push OR eCmd = RudongPump_CMD.Cmd_Pull ) ,pt:=T#20MS);//保证执行的是最新的一次
		IF eCmd = RudongPump_CMD.Cmd_Push
		THEN
			st_IOData.O_DirectionSet := 1	;			
		END_IF
		IF eCmd = RudongPump_CMD.Cmd_Pull 
		THEN
			st_IOData.O_DirectionSet := 0	;			
		END_IF
		IF _tonDelay.Q
		THEN	
			_aExecute[4] := TRUE;//启动夹紧控制数据发送	
			//复位定时器
			_tonDelay(IN:=FALSE);
			_tonCmdTimeout(in:=FALSE);
			_tonTimeout(in:=FALSE);
			_diCmdState := _diCmdState+1;//切换状态
		END_IF
		
	9://等待方向设定被响应
		_tonCmdTimeout(IN:= _aExecute[4],pt:=T#2S);
		IF NOT _aExecute[4]//
		THEN		
			_diCmdState := _diCmdState +1; 
			_tonDelay(IN:=FALSE);
			_tonCmdTimeout(in:=FALSE);
			_tonTimeout(in:=FALSE);
		END_IF	
		IF _tonCmdTimeout.Q
		THEN
			eERRORID := RudongPump_ERROR.FLT_CMD_TIMEOUT;		
			_diCmdState := 999;
		END_IF	
		
	10://重复次数设定		
		_tonDelay(IN:= TRUE,pt:=T#25MS);//保证执行的是最新的一次
		st_IOData.O_CycleNumber := iCycleNumber	;	
		IF _tonDelay.Q
		THEN	
			_aExecute[9] := TRUE;//启动夹紧控制数据发送	
			//复位定时器
			_tonDelay(IN:=FALSE);
			_tonCmdTimeout(in:=FALSE);
			_tonTimeout(in:=FALSE);
			_diCmdState := _diCmdState+1;//切换状态
		END_IF
		
	11://等待重复次数设定被响应
		_tonCmdTimeout(IN:= _aExecute[9],pt:=T#2S);
		IF NOT _aExecute[9]//
		THEN		
			_tonDelay(IN:=TRUE,PT:= T#50MS);
			IF _tonDelay.Q
			THEN
				_tonTimeout(in:=FALSE);
				_tonDelay(IN:=FALSE);
				_tonCmdTimeout(IN:= FALSE); 
				_diCmdState := _diCmdState+1;//切换状态
			END_IF	
		END_IF	
		IF _tonCmdTimeout.Q
		THEN
			eERRORID := RudongPump_ERROR.FLT_CMD_TIMEOUT;		
			_diCmdState := 999;
		END_IF		
		
	12://启动设定		
		_tonDelay(IN:= TRUE ,pt:=T#25MS);//保证执行的是最新的一次	
		st_IOData.O_ControlSet := 1	;					
		IF _tonDelay.Q
		THEN	
			_aExecute[3] := TRUE;//启动夹紧控制数据发送	
			//复位定时器
			_tonDelay(IN:=FALSE);
			_tonCmdTimeout(in:=FALSE);
			_tonTimeout(in:=FALSE);
			_diCmdState := _diCmdState+1;//切换状态
		END_IF
		
	13://等待启动被响应
		_tonTimeout(in:=TRUE,pt:=T#4S); 		
		_tonCmdTimeout(IN:= _aExecute[3],pt:=T#2S);
		IF stPara.xPumpRunSignal//一定要检测到泵运行
		THEN		
			_tonDelay(IN:=FALSE);
			_tonCmdTimeout(in:=FALSE);
			_diCmdState := _diCmdState +1; 
			_tonTimeout(in:=FALSE);	
		END_IF			
		IF _tonCmdTimeout.Q
		THEN
			eERRORID := RudongPump_ERROR.FLT_CMD_TIMEOUT;		
			_diCmdState := 999;
		END_IF
	IF _tonTimeout.Q
  THEN
		_iNGCount := _iNGCount + 1;		
		IF _iNGCount <= 3
		THEN
			_tonDelay(IN:=FALSE);
			_tonCmdTimeout(in:=FALSE);
			_tonTimeout(in:=FALSE);
			_diCmdState := 10;//重新触发启动
		ELSE
			IF eCmd = RudongPump_CMD.Cmd_Push
			THEN
				eERRORID := RudongPump_ERROR.FLT_PUSH_TIMEOUT;		
			END_IF
			IF eCmd = RudongPump_CMD.Cmd_Pull 
			THEN
				eERRORID := RudongPump_ERROR.FLT_PULL_TIMEOUT;			
			END_IF			
			_diCmdState := 999;
		END_IF
	 END_IF	 	
	 
	14://等待运行完成
		_tonTimeout(in:=TRUE,pt:=T#30S); 	
		//夹取成功判定
	 	IF NOT stPara.xPumpRunSignal//电机停止
		THEN
			_tonCmdTimeout(in:=FALSE);
			_tonDelay(IN:= FALSE);
			_tonTimeout(in:=FALSE);  
			_iActRunNumber := _iActRunNumber + 1;
			IF _iActRunNumber >= iCycleNumber//已经到达重复次数
			THEN 
				_diCmdState := 100;
				xComplete := TRUE;
			ELSE
				_diCmdState := 13;
			END_IF
		END_IF		
		IF _tonTimeout.Q//动作超时
		THEN
			IF eCmd = RudongPump_CMD.Cmd_Push
			THEN
				eERRORID := RudongPump_ERROR.FLT_PUSH_TIMEOUT;		
			END_IF
			IF eCmd = RudongPump_CMD.Cmd_Pull 
			THEN
				eERRORID := RudongPump_ERROR.FLT_PULL_TIMEOUT;			
			END_IF			
			_diCmdState := 999;
		END_IF
		
	15://等待下一个周期的启动
		_tonTimeout(in:=TRUE,pt:=T#30S); 				
		//夹取成功判定
		IF stPara.xPumpRunSignal//一定要检测到泵运行
		THEN		
			_tonDelay(IN:=FALSE);
			_tonCmdTimeout(in:=FALSE);
			_tonTimeout(in:=FALSE);
			_diCmdState := _diCmdState - 1; 
		END_IF	
		IF _tonTimeout.Q//动作超时
		THEN
			IF eCmd = RudongPump_CMD.Cmd_Push
			THEN
				eERRORID := RudongPump_ERROR.FLT_PUSH_TIMEOUT;		
			END_IF
			IF eCmd = RudongPump_CMD.Cmd_Pull 
			THEN
				eERRORID := RudongPump_ERROR.FLT_PULL_TIMEOUT;			
			END_IF			
			_diCmdState := 999;
		END_IF	
	ELSE
		;	
END_CASE
END_METHOD

ACTION ConnectAction:
_aWrite_VAR(
			sIPAddr:= stPara.strSlaveIP, 
			nTCPPort:= stPara.iSlavePort, 
			nUnitID:= stPara.bySlaveID, 
			nQuantity:= _aQuantity[_iChannelIndex], 
			nMBAddr:= _aMBAddr[_iChannelIndex], 
			cbLength:= _aQuantity[_iChannelIndex] * 2, 
			pSrcAddr:= ADR(_aAddr[_iChannelIndex,1]), 
			bExecute:=, 
			tTimeout:= T#1000MS, 
			bBusy=> , 
			bError=> , 
			nErrId=> );	

//收发流程管控
CASE _rxState OF 
	0:  _aWrite_VAR.bExecute:=FALSE;
	    _iChannelIndex:=0;
		IF NOT _aWrite_VAR.bBusy //等待功能块触发
		THEN
			_rxState := _rxState + 1;
		END_IF
	1:
		FOR i := 1 TO 15 BY 1//进行读取指令的轮训
		DO
			IF _aExecute[i]//检测有控制指令发生
			THEN 
			    _aWrite_VAR.bExecute:=_aExecute[i]; 
          _iChannelIndex:=i;//触发对应的读写功能		
				IF  _aWrite_VAR.bBusy//只要不是busy状态就代表此时没有指令被响应
				THEN					
					_rxState := _rxState + 1;
				END_IF	
			END_IF
		END_FOR	
		_tonDelay1(in:=FALSE);	
    eMobbusErrorID := 0;	
	2://数据解析	
		FOR i := 1 TO 15 BY 1//进行通用指令轮训
		DO
			IF NOT _aWrite_VAR.bBusy AND NOT _aWrite_VAR.bError  AND _aExecute[i]//对应你功能指令完成
			THEN			 
				_iComNGCount := 0;
				_aExecute[i] := FALSE;
				_aWrite_VAR.bExecute:=FALSE;				
				_rxState := 0;//等待下次触发				
				EXIT;
			END_IF			
			IF _aWrite_VAR.bError AND _aExecute[i]//有错误发生()
			THEN	
				_iComNGCount := _iComNGCount + 1;
				IF _iComNGCount < 3//
        THEN	
				   _aWrite_VAR.bExecute:=FALSE;		
				   _tonDelay1(in:=FALSE);
			     _rxState := _rxState + 1;
				ELSE//					
					 eMobbusErrorID := _aWrite_VAR.nErrid;						
				   _aWrite_VAR.bExecute:=FALSE;					
					 _rxState := 999;//进入错误发生状态	
				END_IF
				EXIT;				
			END_IF			
		END_FOR 
		IF _tonDelay1.Q
		THEN
			_iComNGCount := _iComNGCount + 1;//错误次数加一
			IF _iComNGCount >= 2//重发多次失败
			THEN
					IF _aWrite_VAR.bError 
					THEN
						eMobbusErrorID := _aWrite_VAR.nErrId;						
					END_IF									
				_rxState := 999;//进入错误发生状态
			ELSE
				_tonDelay1(in:=FALSE);
			  _aWrite_VAR.bExecute:=FALSE;
				_rxState:= _rxState + 1;	
			END_IF
		END_IF				
	3://delay
		_tonDelay1(in:=TRUE,PT:=T#60MS);
		IF _tonDelay1.Q
		THEN
			_rxState := 0;
			_tonDelay1(in:=FALSE);	
    END_IF	
	999://错误状态，等待复位发生
		IF _fResetCheck.Q
		THEN
			FOR i:= 1 TO 15 DO
				_aExecute[i] := FALSE;
				_aWrite_VAR.bExecute:=FALSE;					
			END_FOR		
			_iComNGCount := 0;//
			_rxState := 0;//重新开始			
		END_IF
	ELSE
		;
END_CASE
END_ACTION

METHOD PROTECTED CyclicAction
VAR_INPUT
END_VAR
VAR_OUTPUT
	xComplete: BOOL;
END_VAR
VAR	
END_VAR
IF xAbort=0 THEN
    IF xFirstInvocation THEN
    (*
    * Staring
    * for then first (!) invocaion,
    * sample then input variables
    *)			
    _diCmdState:= 0;
	_iNGCount := 0;
	_iActRunNumber := 0;
	xFirstInvocation:=0;			
    END_IF    
    REPEAT 				
		  (**************************检查是否有硬件报错(检测总线是否报错)**********************************) 
			IF _xConnectError
			THEN
				eERRORID := RudongPump_ERROR.FLT_CONNECT;//子站通讯报警
			END_IF
			//检测参数是否配置正确	
			IF ( stPara.iType <> 1 AND stPara.iType <> 2 )//只能是modbus模式	 
			THEN
				eERRORID := RudongPump_ERROR.FLT_PARA;//参数配置错误
			END_IF
	
			//检测停止指令是否发生
			_rStopCmdTrig(CLK:= NOT xEStop OR (stDeviceOpe.xStop_Hmi AND NOT xAutoMode AND NOT xDeviceRunning) OR (stDeviceOpe.xStop_Auto AND (xAutoMode OR xDeviceRunning))
													OR (stDeviceOpe.xFullSpeedStop_Hmi AND NOT xAutoMode AND NOT xDeviceRunning) OR (stDeviceOpe.xFullSpeedStop_Auto AND (xAutoMode OR xDeviceRunning)));		
		  IF _rStopCmdTrig.Q//检测到停止指令
			THEN
				_diCmdState := 0;
				eCmd := RudongPump_CMD.Cmd_Stop;
				_tonCmdTimeout(in:=FALSE);
				_tonDelay(IN:= FALSE);
				_tonTimeout(in:=FALSE);
			END_IF			
			//检测是否有Modbus指令运行中	
			_xCheckModbusRun := FALSE;
			FOR i:=0 TO 14 BY 1 
			DO 
				_xCheckModbusRun := _aWrite_VAR.bBusy OR _aExecute[i];
			END_FOR		
		
			CASE eCmd OF//判断指令类型
				RudongPump_CMD.Cmd_Pull,RudongPump_CMD.Cmd_Push://执行夹爪指令(夹紧和松开指令)
					CmdRunAction(xComplete=> xComplete);	
							
				RudongPump_CMD.Cmd_Stop,RudongPump_CMD.Cmd_FullSpeedStop://执行过程中等待停止指令(分为运行停止和全速停止)
					mCmdStopAction(xComplete=> xComplete);
					
				RudongPump_CMD.Cmd_Configure://(用于配置参数)
					mCmdConfigureAction(xComplete=> xComplete);
					
				RudongPump_CMD.Cmd_FullSpeedPush,RudongPump_CMD.Cmd_FullSpeedPull://全速启动控制（用于清洗和充满试管）
					mCmdFullSpeedStartAction(xComplete=> xComplete);
					
				RudongPump_CMD.Cmd_CalPump:
					CmdPumpCal(xComplete=> xComplete);

				RudongPump_CMD.Cmd_CalReset:
					CmdCalReset(xComplete=> xComplete);			
				ELSE
					;	
				END_CASE		   
      UNTIL (TRUE)
	END_REPEAT
END_IF

IF xAbort OR xComplete OR eERRORID<>RudongPump_ERROR.No_ERROR THEN    
    (*
    * Cleaning
    * => free as much allocated resources as possible
    *)    
    tOperationTimer(IN:=0);
END_IF
END_METHOD

METHOD PRIVATE FINAL HandleAbortedState
VAR_INPUT
END_VAR
VAR_OUTPUT
	xAgain: BOOL;
END_VAR
VAR
	xComplete: BOOL;
END_VAR
IF xAborted AND xResetRequest THEN
    eState:=STATE.RESETING;
    xAgain:=1;
ELSE
    xBusy:=0;
    xAborted:=1;
    //xResetRequest:=(xExecute=0);
    xAgain:=0;(* !!! *)
END_IF
END_METHOD

METHOD PRIVATE FINAL HandleAbortingState
VAR_INPUT
END_VAR
VAR_OUTPUT
	xAgain: BOOL;
END_VAR
VAR
	xComplete: BOOL;
END_VAR
AbortAction(xComplete=> xComplete, eERRORID=> eERRORID);

IF eERRORID<>RudongPump_ERROR.No_ERROR THEN
    eState:=STATE.INERROR;
    xAgain:=1;
ELSIF xComplete THEN
    eState:=STATE.ABORTED;
    xAgain:=1;
END_IF
END_METHOD

METHOD PRIVATE FINAL HandleDoneState
VAR_INPUT
END_VAR
VAR_OUTPUT
	xAgain: BOOL;
END_VAR
//在运行过程中要是切换模式，再运行完成之后，检测到模式的切换，就需要回到初始位置，进行下一次执行准备
IF _xDone AND ((xExecute=0) OR ( _xModeChange AND NOT _xAutoOpe)  OR ( NOT xAutoMode AND NOT xDeviceRunning AND ( NOT _xAutoOpe OR _xHMIOpe))) THEN
	eState:=STATE.RESETING;
	xAgain:=1;
ELSE
	xBusy:=0;
	_xDone:=1;
	xAgain:=0;(* !!! *)
END_IF
END_METHOD

METHOD PRIVATE FINAL HandleDormantState
VAR_INPUT
END_VAR
VAR_OUTPUT
	xAgain: BOOL;
END_VAR
IF xExecute THEN
    xBusy:=1;
    eState:=STATE.EXECUTING;
    xAgain:=1;
END_IF
//下面两个报警一旦报警就需要发生
IF _xConnectError 
THEN//出现这个进行报警
	eERRORID := RudongPump_ERROR.FLT_CONNECT;//子站通讯报警
END_IF

IF _fResetCheck.Q//清空报警
THEN
	eERRORID := RudongPump_ERROR.No_ERROR;
END_IF
IF  xAutoMode OR xDeviceRunning THEN
	xAutomodeFlag:=TRUE;
ELSE
	xAutomodeFlag:=FALSE;
END_IF


IF eErrorID = RudongPump_ERROR.NO_ERROR 
THEN
	IF   xRunILC   THEN
		FOR k:=1 TO 5 BY 1 DO
			//PULL
			_rOperaTrig[k](CLK:=xRunILC AND (stDeviceOpe.xPull_Hmi[k] AND NOT xAutomodeFlag) OR (stDeviceOpe.xPull_Auto[k] AND xAutomodeFlag));
			IF _rOperaTrig[k].Q //
			THEN
				rFluVolumeSet	:=stRunPara.rPullFluVolume[k];
				rRuntimeSet		:=stRunPara.rPullRuntime[k];
				iCycleNumber	:=stRunPara.iPullCycleNumber[k];
				eCmd 			:= RudongPump_CMD.Cmd_Pull;
				xExecute		:= TRUE;
			END_IF		
			//PUSH
			_rOperaTrig[k+5](CLK:=xRunILC AND (stDeviceOpe.xPush_Hmi[k] AND NOT xAutomodeFlag) OR (stDeviceOpe.xPush_Auto[k] AND xAutomodeFlag));
			IF _rOperaTrig[k+5].Q 
			THEN
				rFluVolumeSet	:=stRunPara.rPushFluVolume[k];  
				rRuntimeSet		:=stRunPara.rPushRuntime[k];    
				iCycleNumber	:=stRunPara.iPushCycleNumber[k];
				eCmd 			:= RudongPump_CMD.Cmd_Push;
				xExecute 		:= TRUE;
			END_IF				
		END_FOR
		//STOP
		 IF(stDeviceOpe.xStop_Hmi AND  NOT xAutomodeFlag) OR NOT xEStop OR stDeviceOpe.xStop_Auto    THEN
				eCmd := RudongPump_CMD.Cmd_Stop;
				xExecute := TRUE;
		 END_IF
		//FullSpeedPull
		IF (stDeviceOpe.xFullSpeedPull_Hmi AND  NOT xAutomodeFlag) OR (stDeviceOpe.xFullSpeedPull_Auto AND  xAutomodeFlag) THEN
			eCmd := RudongPump_CMD.Cmd_FullSpeedPull;
			xExecute := TRUE;
		END_IF
		//FullSpeedPush
		IF (stDeviceOpe.xFullSpeedPush_Hmi AND NOT xAutomodeFlag ) OR (stDeviceOpe.xFullSpeedPush_Auto AND xAutomodeFlag) THEN	
			eCmd := RudongPump_CMD.Cmd_FullSpeedPush;
			xExecute := TRUE;
		END_IF
		//FullSpeedStop
		 IF (stDeviceOpe.xFullSpeedStop_Hmi AND NOT xAutomodeFlag) OR (stDeviceOpe.xFullSpeedStop_Auto AND xAutomodeFlag) THEN	
			eCmd := RudongPump_CMD.Cmd_FullSpeedStop;
			xExecute := TRUE;
		END_IF
		//Configure
		IF (stDeviceOpe.xConfigure_Hmi AND NOT xAutomodeFlag) OR (stDeviceOpe.xConfigure_Auto AND xAutomodeFlag) THEN	
			eCmd := RudongPump_CMD.Cmd_Configure;
			xExecute := TRUE;
		END_IF
		
	END_IF		
		//校准
		IF stDeviceOpe.xPumpCal_Hmi OR stDeviceOpe.xPumpCal_Auto THEN
			rFluVolumeSet		:=stRunPara.rCalFluVolume;
			rRuntimeSet			:=stRunPara.rCalTime;
			iCycleNumber		:=stRunPara.rCalNum;	
			iModuleAdress		:=stRunPara.iModuleAdress;
			iModuleSpeed		:=stRunPara.rModuleSpeed;
			iModuleRealVolume	:=stRunPara.rModuleRealFluVolume;		
			eCmd 				:= RudongPump_CMD.Cmd_CalPump;
			xExecute 			:= TRUE;		
		END_IF
		
		//复位校准系数为初始值
		IF stDeviceOpe.xResetCalcoeffCal_Hmi THEN	
			eCmd 				:= RudongPump_CMD.Cmd_CalReset;
			xExecute 			:= TRUE;		
		END_IF
	
				
END_IF
END_METHOD

METHOD PRIVATE FINAL  HandleErrorState
VAR_INPUT
END_VAR
VAR_OUTPUT
	xAgain: BOOL;
END_VAR
IF xRudongPump_ERROR AND  (xResetRequest OR NOT xExecute) THEN
    eState:=STATE.RESETING;
    xAgain:=1;
ELSE
    xBusy:=0;
    xRudongPump_ERROR:=1;    
    xAgain:=0;(* !!! *)
END_IF
END_METHOD

METHOD PRIVATE FINAL HandleExecutingState
VAR_INPUT
END_VAR
VAR_OUTPUT
	xAgain: BOOL;
END_VAR
VAR
	xComplete: BOOL;
END_VAR
IF xAbort=0 THEN   
    CyclicAction(xComplete=> xComplete);
END_IF

IF eERRORID<>RudongPump_ERROR.No_ERROR THEN
    eState:=STATE.INERROR;
    xAgain:=1;
ELSIF xAbort THEN
    eState:=STATE.ABORTING;
    xAgain:=1;
ELSIF xComplete THEN
    eState:=STATE.DONE;
    xAgain:=1;
END_IF
END_METHOD

METHOD PRIVATE FINAL HandleResettingState
VAR_INPUT
END_VAR
VAR_OUTPUT
	xAgain: BOOL;
END_VAR
VAR
	xComplete: BOOL;
END_VAR
ResetAction(xComplete=> xComplete);

IF xComplete THEN
	xExecute:=0;//清除输入指令 
    xBusy:=0;
    _xDone:=0;
    xRudongPump_ERROR:=0;
    xAborted:=0;
    eERRORID:=RudongPump_ERROR.No_ERROR;
    eState:=STATE.DORMANT;
    xFirstInvocation:=1;
    xAgain:=0;(* !!! *)
END_IF
END_METHOD

METHOD PROTECTED mCmdConfigureAction
VAR_OUTPUT
	xComplete: BOOL;
END_VAR
VAR
END_VAR
// return the real actual fault number
IF eERRORID <> RudongPump_ERROR.No_ERROR
THEN
  RETURN;  
END_IF

CASE _diCmdState OF
	0://使能失效操作	
		IF _xConfigureParaOK THEN
			st_IOData.O_PumpType := stRunPara.iPumpTypeSet;
			_tonDelay(IN:=TRUE,PT:=T#25MS);
			IF _tonDelay.Q//等待指令响应
			THEN
				_aExecute[1] := TRUE;//触发运行指令	
				//复位定时器
				_tonTimeout(in:=FALSE);
				_tonDelay(IN:=FALSE);
				_tonCmdTimeout(IN:= FALSE);    
				_diCmdState := _diCmdState+1;//切换状态
			END_IF	
		ELSE//输入配置参数错误
			eERRORID := RudongPump_ERROR.FLT_CONFIGURE_PARA;	
			diStepOld:=	_diCmdState;
			_diCmdState := 999;
		END_IF		  		

	1://等待使能失效被响应	
		_tonCmdTimeout(IN:= TRUE,pt:=T#2S);
		IF NOT _aExecute[1]
		THEN
			_tonDelay(IN:=TRUE,PT:= T#50MS);
			IF _tonDelay.Q
			THEN			
				_tonTimeout(in:=FALSE);
				_tonDelay(IN:=FALSE);
				_tonCmdTimeout(IN:= FALSE);    
				_diCmdState := _diCmdState+1;//切换状态
			END_IF			
		END_IF	
		IF _tonCmdTimeout.Q//指令超时报错
		THEN
			eERRORID := RudongPump_ERROR.FLT_CMD_TIMEOUT;	
			diStepOld:=	_diCmdState;	
			_diCmdState := 999;
		END_IF	
	2://设置软管类型		
		st_IOData.O_HosePipeType := stRunPara.iHosePipeTypeSet;
		_tonDelay(IN:=TRUE,PT:=T#25MS);
		IF _tonDelay.Q//等待指令响应
		THEN
			_aExecute[2] := TRUE;//触发运行指令	
			//复位定时器
			_tonTimeout(in:=FALSE);
			_tonDelay(IN:=FALSE);
			_tonCmdTimeout(IN:= FALSE);    
			_diCmdState := _diCmdState+1;//切换状态
		END_IF	
	3://等待使能失效被响应	
		_tonCmdTimeout(IN:= TRUE,pt:=T#2S);
		IF NOT _aExecute[2]
		THEN
			_tonCmdTimeout(in:=FALSE);
			_tonDelay(IN:= FALSE);
			_tonTimeout(in:=FALSE);  
			_diCmdState := 100;
			 xComplete := 1;
		END_IF	
		IF _tonCmdTimeout.Q//指令超时报错
		THEN
			eERRORID := RudongPump_ERROR.FLT_CMD_TIMEOUT;
			diStepOld:=	_diCmdState;		
			_diCmdState := 999;
		END_IF	 
	ELSE
		;
END_CASE
END_METHOD

METHOD PROTECTED mCmdFullSpeedStartAction
VAR_OUTPUT
	xComplete: BOOL;
END_VAR
VAR
END_VAR
// return the real actual fault number
IF eERRORID <> RudongPump_ERROR.No_ERROR
THEN
  RETURN;  
END_IF

CASE _diCmdState OF
	0://方向设定		
		_tonDelay(IN:= ( eCmd = RudongPump_CMD.Cmd_FullSpeedPush OR eCmd = RudongPump_CMD.Cmd_FullSpeedPull ) ,pt:=T#20MS);//保证执行的是最新的一次
		IF eCmd = RudongPump_CMD.Cmd_FullSpeedPush
		THEN
			st_IOData.O_DirectionSet := 1	;			
		END_IF
		IF eCmd = RudongPump_CMD.Cmd_FullSpeedPull 
		THEN
			st_IOData.O_DirectionSet := 0	;			
		END_IF
		IF _tonDelay.Q
		THEN	
			_aExecute[4] := TRUE;//启动夹紧控制数据发送	
			//复位定时器
			_tonDelay(IN:=FALSE);
			_tonCmdTimeout(in:=FALSE);
			_tonTimeout(in:=FALSE);
			_diCmdState := _diCmdState+1;//切换状态
		END_IF
			
	1://等待方向设定被响应
		_tonCmdTimeout(IN:= _aExecute[4],pt:=T#2S);
		IF NOT _aExecute[4]//
		THEN		
			_tonDelay(IN:=TRUE,PT:= T#50MS);
			IF _tonDelay.Q
			THEN			
				_tonTimeout(in:=FALSE);
				_tonDelay(IN:=FALSE);
				_tonCmdTimeout(IN:= FALSE);    
				_diCmdState := _diCmdState+1;//切换状态
			END_IF	
		END_IF	
		IF _tonCmdTimeout.Q
		THEN
			eERRORID := RudongPump_ERROR.FLT_CMD_TIMEOUT;		
			_diCmdState := 999;
		END_IF	
	2://使能失效操作		     
		st_IOData.O_FullSpeedControl := 1;		
		_tonDelay(IN:=TRUE,PT:=T#25MS);
		IF _tonDelay.Q//等待指令响应
		THEN
			_aExecute[5] := TRUE;//触发运行指令	
			//复位定时器
			_tonTimeout(in:=FALSE);
			_tonDelay(IN:=FALSE);
			_tonCmdTimeout(IN:= FALSE);    
			_diCmdState := _diCmdState+1;//切换状态
		END_IF
	3://等待使能失效被响应	
		_tonCmdTimeout(IN:= TRUE,pt:=T#2S);
		IF NOT _aExecute[5] 
		THEN
			_tonCmdTimeout(in:=FALSE);
			_tonDelay(IN:= FALSE);
			_tonTimeout(in:=FALSE);  
			_diCmdState := 100;
			 xComplete := 1; 
		END_IF	
		IF _tonCmdTimeout.Q//指令超时报错
		THEN
			eERRORID := RudongPump_ERROR.FLT_CMD_TIMEOUT;		
			_diCmdState := 999;
		END_IF		
	ELSE
		;
END_CASE
END_METHOD

METHOD PROTECTED mCmdStopAction
VAR_OUTPUT
	xComplete: BOOL;
END_VAR
VAR
END_VAR
// return the real actual fault number
IF eERRORID <> RudongPump_ERROR.No_ERROR
THEN
  RETURN;  
END_IF

CASE _diCmdState OF
	0://使能失效操作
		st_IOData.O_ControlSet := 0;
		st_IOData.O_FullSpeedControl := 0;		  
		_tonDelay(IN:=TRUE,PT:=T#25MS);
		IF _tonDelay.Q//等待指令响应
		THEN
			IF eCmd = RudongPump_CMD.Cmd_Stop
			THEN
				_aExecute[3] := TRUE;//触发运行指令	
			END_IF
			IF eCmd = RudongPump_CMD.Cmd_FullSpeedStop
			THEN
				_aExecute[5] := TRUE;//触发运行指令	
			END_IF
			//复位定时器
			_tonTimeout(in:=FALSE);
			_tonDelay(IN:=FALSE);
			_tonCmdTimeout(IN:= FALSE);    
			_diCmdState := _diCmdState+1;//切换状态
		END_IF			

	1://等待使能失效被响应	
		_tonCmdTimeout(IN:= TRUE,pt:=T#2S);
		IF NOT _aExecute[3] AND  NOT _aExecute[5]
		THEN
			_tonCmdTimeout(in:=FALSE);
			_diCmdState := _diCmdState +1; 
		END_IF	
		IF _tonCmdTimeout.Q//指令超时报错
		THEN
			eERRORID := RudongPump_ERROR.FLT_CMD_TIMEOUT;		
			_diCmdState := 999;
		END_IF	
  2://延时100ms错开信号
		_tonDelay(IN:= TRUE,pt:=T#100MS);//设置刷新周期
		IF _tonDelay.Q
		THEN			
			_diCmdState := _diCmdState + 1;
		END_IF		 		
	3://等待数据接收完成		
		_tonTimeout(in:=TRUE,pt:=T#10S);//设置超时时间	
		IF NOT stPara.xPumpRunSignal  //代表电机已经停机
		THEN
			_tonCmdTimeout(in:=FALSE);
			_tonDelay(IN:= FALSE);
			_tonTimeout(in:=FALSE);  
			_diCmdState := 100;
			xComplete := 1;
		END_IF		
		IF _tonTimeout.Q//回原点动作超时，或者回原点报错
		THEN
			IF eCmd = RudongPump_CMD.Cmd_Stop
				THEN
					eERRORID := RudongPump_ERROR.FLT_STOP_TIMEOUT;
				END_IF
				IF eCmd = RudongPump_CMD.Cmd_FullSpeedStop
				THEN
					eERRORID := RudongPump_ERROR.FLT_FULLSPEEDSTOP_TIMEOUT;
				END_IF			
			_diCmdState := 999;
		END_IF	
	ELSE
		;
END_CASE
END_METHOD

METHOD PROTECTED ResetAction
VAR_INPUT
END_VAR
VAR_OUTPUT
	xComplete: BOOL;
END_VAR
(*
* Cleaning
* => free all allocated resources
* => reinitialize instance variables
*)
tOperationTimer(IN:=0);
tInvocationTimer(IN:=0);

// init command state
_diCmdState := 0;
_tonCmdTimeout(in:=FALSE);
_tonDelay(IN:= FALSE);
_tonTimeout(in:=FALSE);
_xModeChange := FALSE;
_rStopCmdTrig(CLK:=FALSE);
_iNGCount := 0;

//清除触发标志位
FOR i:=1 TO 15 BY 1 
DO 
	_aExecute[i] := FALSE;
	_aWrite_VAR.bExecute := FALSE;	
END_FOR
//清除触发状态
FOR k:=1 TO 15 BY 1 DO
	_rOperaTrig[k](CLK:=FALSE);
END_FOR	
	
stDeviceOpe.xConfigure_Auto:= stDeviceOpe.xConfigure_Hmi:= FALSE;
stDeviceOpe.xStop_Auto:= stDeviceOpe.xStop_Hmi:= FALSE;
stDeviceOpe.xFullSpeedPull_Auto:= stDeviceOpe.xFullSpeedPull_Hmi:= FALSE;
stDeviceOpe.xFullSpeedPush_Auto:= stDeviceOpe.xFullSpeedPush_Hmi:= FALSE;
stDeviceOpe.xFullSpeedStop_Auto:= stDeviceOpe.xFullSpeedStop_Hmi:= FALSE;
FOR k:=1 TO 5 DO
	stDeviceOpe.xPull_Auto[k]:= stDeviceOpe.xPull_Hmi[k] := FALSE;
	stDeviceOpe.xPush_Auto[k]:= stDeviceOpe.xPush_Hmi[k] := FALSE;
END_FOR

stDeviceOpe.xPumpCal_Auto:=stDeviceOpe.xPumpCal_Hmi:=FALSE;
stDeviceOpe.xResetCalcoeffCal_Hmi:=FALSE;
st_IOData.O_ModuleStart := 0	;
xResetRequest:=FALSE;
//复位完成
xComplete:=1;
END_METHOD

END_FUNCTION_BLOCK

// ---- POUs/40_TcpIp/40_TcpIp/FB_ClientDataExcha.TcPOU
{attribute 'tc_no_symbol'}
FUNCTION_BLOCK FB_ClientDataExcha
VAR_INPUT
	hSocket				: T_HSOCKET;
	aToServer			: ARRAY[1..MAX_PLCPRJ_RXBUFFER_SIZE] OF BYTE;//发送数据缓存区
	udiSendNumber : UDINT;
	xEnable: BOOL;//使能失效标志位
	xResetRequest: BOOL;   
	dwTimeOut: DWORD;//[ms],0 => no executing time limit
	xNeedReceive : BOOL;//检测是否需要接收标志位
	xReceiveAlways : BOOL ;//检测是否需要一直进行读取
END_VAR
VAR_OUTPUT
	xRdyCmd : BOOL;(*是否满足接收指令*)
	xDone: BOOL;(*完成条件满足*)
	xBusy: BOOL;(*动作正在执行*)
	xError: BOOL;(*错误条件满足*)
	udiErrorID: UDINT;(*错误码*)
	sFromServer		: T_MaxString;//实际接收数据(字符串)
	rxBuffer				: ARRAY[1..MAX_PLCPRJ_RXBUFFER_SIZE] OF BYTE;//接收缓存区域(byte数组)
END_VAR
VAR
{attribute 'tc_no_symbol'}
	eState: STATE;//当前状态
{attribute 'tc_no_symbol'}
	eClientState : E_ClientSteps;
{attribute 'tc_no_symbol'}
	xFirstInvocation: BOOL := TRUE;
{attribute 'tc_no_symbol'}	 
	xTimeOut: BOOL;
{attribute 'tc_no_symbol'}
	tOperationTimer : TON;
{attribute 'tc_no_symbol'}	
	fbSocketSend		: FB_SocketSend := ( tTimeout := PLCPRJ_RECEIVE_TIMEOUT );
{attribute 'tc_no_symbol'}
	fbSocketReceive		: FB_SocketReceive := ( tTimeout := PLCPRJ_RECEIVE_TIMEOUT );
{attribute 'tc_no_symbol'}
	fbReceiveTON		: TON;
{attribute 'tc_no_symbol'}	
	fbDisconnectTON		: TON;
{attribute 'tc_no_symbol'}
	RisingEdge			: R_TRIG;
{attribute 'tc_no_symbol'}	
	eDataExchaStep	: E_DataExchaSteps;
{attribute 'tc_no_symbol'}	
	cbReceived , idx	: UDINT;	
{attribute 'tc_no_symbol'}	
	_rxBufferTemp				: ARRAY[1..MAX_PLCPRJ_RXBUFFER_SIZE] OF BYTE;//接收缓存区域
{attribute 'tc_no_symbol'}	
_ton : TON;
END_VAR
VAR_TEMP
{attribute 'tc_no_symbol'}
	xAgain: BOOL;
END_VAR

xAgain:=0;

REPEAT
	CASE eState OF
		STATE.DORMANT:
				HandleDormantState(xAgain=> xAgain);
		STATE.EXECUTING:
				HandleExecutingState(xAgain=> xAgain);
		STATE.DONE:
				HandleDoneState(xAgain=> xAgain);
		STATE.INERROR:
				HandleErrorState(xAgain=> xAgain);
		STATE.ABORTING:
				HandleAbortingState(xAgain=> xAgain);
		STATE.RESETING:
				HandleResettingState(xAgain=> xAgain);
    END_CASE
UNTIL (xAgain=0)
END_REPEAT

xRdyCmd := 	eState = STATE.DORMANT;//输出是否已经准备好响应指令

{attribute 'tc_no_symbol'}
METHOD PROTECTED AbortAction
VAR_INPUT
END_VAR
VAR_OUTPUT
	xComplete: BOOL;
  udiErrorID: UDINT;
END_VAR
(*
* Cleaning
* => abort all running operation
* => if an UDINT codition is reached, set udiErrorID to a Value rather then 0 
*)
xComplete:=1;
udiErrorID:=0;
END_METHOD

{attribute 'tc_no_symbol'} 
METHOD PROTECTED CyclicAction
VAR_INPUT
END_VAR
VAR_OUTPUT
	xComplete: BOOL;
	udiErrorID: UDINT;
END_VAR
VAR	
END_VAR
{attribute 'tc_no_symbol'}
IF xFirstInvocation THEN
(*
* Staring
* for then first (!) invocaion,
* sample then input variables
*)		
	eDataExchaStep := DATAEXCHA_STATE_IDLE;
	xFirstInvocation:=0;			
END_IF    
REPEAT 	 
	CASE eDataExchaStep OF		
		DATAEXCHA_STATE_IDLE:						
			cbReceived := 0; // TODO. Leslie
			fbReceiveTON( IN := FALSE, PT := T#0s ); (* don't wait, read the first answer data immediately *)
			fbDisconnectTON( IN := FALSE, PT := T#0s );(* disable timeout check first *)
			eDataExchaStep := DATAEXCHA_STATE_SEND_START;
	   
		DATAEXCHA_STATE_SEND_START:
			fbSocketSend( bExecute := FALSE );
			fbSocketSend( 	hSocket	:= hSocket,
						cbLen	:= udiSendNumber,(* string length inclusive zero delimiter *)				
						pSrc	:= ADR( aToServer ),
						bExecute:= TRUE );//启动发送			
			eDataExchaStep := DATAEXCHA_STATE_SEND_WAIT;
	
		DATAEXCHA_STATE_SEND_WAIT:
			fbSocketSend( bExecute := FALSE );
			IF NOT fbSocketSend.bBusy THEN//检测发送是否完成
				IF NOT fbSocketSend.bError THEN	
					IF xNeedReceive
					THEN
						fbDisconnectTON(IN := FALSE);
						eDataExchaStep := DATAEXCHA_STATE_RECEIVE_START;							
					ELSE
						SysMemSet( ADR(sFromServer), 0, SIZEOF(sFromServer));		
						eDataExchaStep := DATAEXCHA_STATE_IDLE;		
						xComplete := 1;	
					END_IF	
				ELSE		
					udiErrorID := fbSocketSend.nErrId;								
				END_IF						
			END_IF		
	
		DATAEXCHA_STATE_RECEIVE_START:
			fbDisconnectTON(IN := TRUE,PT:=T#10MS);
			fbSocketReceive(bExecute := FALSE);		
			 
			fbSocketReceive(  hSocket:= hSocket,
											cbLen:= SIZEOF( _rxBufferTemp ),
											pDest:= ADR( _rxBufferTemp),
											bExecute:= TRUE ,
											nRecBytes=>cbReceived); 
      IF fbDisconnectTON.Q
			THEN
				eDataExchaStep := DATAEXCHA_STATE_RECEIVE_WAIT;
				fbDisconnectTON(IN:=FALSE);       
			END_IF
		DATAEXCHA_STATE_RECEIVE_WAIT:	
			_ton(IN:= NOT _ton.Q, PT:= T#20MS, Q=> , ET=> );
			fbSocketReceive(bExecute := _ton.Q,
                      nRecBytes=>cbReceived);	
      fbSocketReceive(bExecute := FALSE);				
			IF NOT fbSocketReceive.bBusy THEN
				IF NOT fbSocketReceive.bError THEN 						
					IF cbReceived < 255 AND cbReceived > 0 THEN(* no overflow *)
						fbReceiveTON( PT := T#0s ); (* bytes received => increase the read (polling) speed *)
						fbDisconnectTON( IN := FALSE );(* bytes received => disable timeout check *)		
						SysMemSet( ADR(sFromServer), 0, SIZEOF(sFromServer));		
						SysMemSet( ADR(rxBuffer), 0, SIZEOF(rxBuffer));	
						SysMemCpy( ADR( rxBuffer ), ADR( _rxBufferTemp ), cbReceived );//进行数据迁移
						SysMemCpy( ADR( sFromServer ), ADR( _rxBufferTemp ), cbReceived );(* copy the received string to the output variable (inclusive the end delimiter) *)								
						eDataExchaStep := DATAEXCHA_STATE_IDLE;		
						xComplete := 1;
					END_IF
					IF cbReceived >= 255(* there is no more free read buffer space => the answer string should be terminated *)	
          THEN
						udiErrorID :=100;(* buffer overflow !*)				
					END_IF			
				ELSE(* receive UDINT *)
					udiErrorID := fbSocketReceive.nErrId;	
				END_IF
			END_IF
			fbDisconnectTON( IN := TRUE, PT := PLCPRJ_RECEIVE_TIMEOUT );(* no bytes received => enable timeout check*)
			IF fbDisconnectTON.Q THEN (* timeout UDINT*)
				fbDisconnectTON( IN := FALSE );
				udiErrorID := 101;//接收超时报错			
			END_IF
		ELSE
			;
	END_CASE	       
UNTIL (TRUE)//让程序一直处于刷新状态
END_REPEAT

IF NOT xEnable OR xComplete OR udiErrorID<>0 THEN    
    (*
    * Cleaning
    * => free as much allocated resources as possible
    *)    
    tOperationTimer(IN:=0);
END_IF
END_METHOD

{attribute 'tc_no_symbol'}
METHOD PRIVATE FINAL HandleAbortingState
VAR_INPUT
END_VAR
VAR_OUTPUT
	xAgain: BOOL;
END_VAR
VAR
{attribute 'tc_no_symbol'}	
	xComplete: BOOL;
END_VAR
AbortAction(xComplete=> xComplete, udiErrorID=> udiErrorID);

IF udiErrorID<>0 THEN
    eState:=STATE.INERROR;
    xAgain:=1;
ELSIF xComplete THEN
    eState:=STATE.INERROR;
    xAgain:=1;
END_IF
END_METHOD

{attribute 'tc_no_symbol'}
METHOD PRIVATE FINAL HandleDoneState
VAR_INPUT
END_VAR
VAR_OUTPUT
	xAgain: BOOL;
END_VAR
IF xDone AND (xEnable=0) THEN
	eState:=STATE.RESETING;
	xAgain:=1;
ELSE
	xBusy:=0;
	xDone:=1;
	//xResetRequest:=(xExecute=0);
	xAgain:=0;(* !!! *)
END_IF
END_METHOD

{attribute 'tc_no_symbol'}
METHOD PRIVATE FINAL HandleDormantState
VAR_INPUT
END_VAR
VAR_OUTPUT
	xAgain: BOOL;
END_VAR
IF xEnable THEN
    xBusy:=1;
    eState:=STATE.EXECUTING;
    xAgain:=1;
END_IF
END_METHOD

{attribute 'tc_no_symbol'}
METHOD PRIVATE FINAL  HandleErrorState
VAR_INPUT
END_VAR
VAR_OUTPUT
	xAgain: BOOL;
END_VAR
IF xError AND (xResetRequest OR NOT xEnable ) THEN
    eState:=STATE.RESETING;
    xAgain:=1;
ELSE
    xBusy:=0;
    xError:=1;    
    xAgain:=0;(* !!! *)
END_IF
END_METHOD

{attribute 'tc_no_symbol'}
METHOD PRIVATE FINAL HandleExecutingState
VAR_INPUT
END_VAR
VAR_OUTPUT
	xAgain: BOOL;
END_VAR
VAR
{attribute 'tc_no_symbol'}	
	xComplete: BOOL;
END_VAR
 
CyclicAction(xComplete=> xComplete, udiErrorID=> udiErrorID);


IF udiErrorID<>0 THEN//检测是否有错误发生
    eState:=STATE.INERROR;
    xAgain:=1;
ELSIF NOT xEnable THEN//检测使能条件
    eState:=STATE.ABORTING;
    xAgain:=1;
ELSIF xComplete THEN//检测是否正常处理完成
    eState:=STATE.DONE;
    xAgain:=1;
END_IF
END_METHOD

{attribute 'tc_no_symbol'}
METHOD PRIVATE FINAL HandleResettingState
VAR_INPUT
END_VAR
VAR_OUTPUT
	xAgain: BOOL;
END_VAR
VAR
{attribute 'tc_no_symbol'}
	xComplete: BOOL;
END_VAR
ResetAction(xComplete=> xComplete);

IF xComplete THEN
		xEnable:=0;//清除输入指令 
    xBusy:=0;
    xDone:=0;
    xError:=0;

    udiErrorID:=0;
    eState:=STATE.DORMANT;
    xFirstInvocation:=1;
    xAgain:=0;(* !!! *)
END_IF
END_METHOD

{attribute 'tc_no_symbol'}
METHOD PROTECTED ResetAction
VAR_INPUT
END_VAR
VAR_OUTPUT
	xComplete: BOOL;
END_VAR
(*
* Cleaning
* => free all allocated resources
* => reinitialize instance variables
*)
tOperationTimer(IN:=0);

fbSocketSend( bExecute := FALSE );
fbSocketReceive(bExecute := FALSE);		

eDataExchaStep := DATAEXCHA_STATE_IDLE;		

xComplete := 1;
END_METHOD

END_FUNCTION_BLOCK
